{attribute 'qualified_only'}
TYPE E_OpMod_Binary :
(
	eOff			:= 0,
	eOn				:= 1
	
) UDINT;
END_TYPE

(* stored: Version 1.1.0.1, ProductVersion 3.1.4024.5
   DUT E_OpMod_Binary: Id {f1158d08-f38d-4cd7-ac6e-87677e274444} *)
